// TIA Portal V17 export
// export: Created 2024-08-26T21:10:51.7294849Z, ExportSetting WithDefaults, DisplayName Totally Integrated Automation Portal, DisplayVersion V17 Update 7, DisplayName TIA Portal Openness, DisplayVersion V17 Update 7, DisplayName TIA Portal Version Control Interface, DisplayVersion V17, DisplayName SINAMICS Startdrive Advanced, DisplayVersion V17 SP2, DisplayName SINAMICS Startdrive G110M, G120, G120C, G120D, G120P, G115D, DisplayVersion V17 SP2, DisplayName SINAMICS Startdrive G130, G150, S120, S150, SINAMICS MV, S210, DisplayVersion V17 SP2, DisplayName STEP 7 Professional, DisplayVersion V17 Update 7, DisplayName STEP 7 Safety, DisplayVersion V17 Update 6, DisplayName WinCC Advanced / Unified PC, DisplayVersion V17 Update 7
DATA_BLOCK "DB_MODEL"   // DB5
{ S7_Optimized_Access := 'TRUE' }
VERSION : 0.1
// stored: AutoNumber false, DBAccessibleFromOPCUA true, DBAccessibleFromWebserver true, IsOnlyStoredInLoadMemory false, IsRetainMemResEnabled false, IsWriteProtectedInAS false, MemoryReserve 100
   VAR RETAIN
      "name" : Array[0..32] of String[50];
   END_VAR
   VAR
      day : Int := 6;
      dayText : String := '    11';
      month : Int := 8;
      monthText : String := '     8';
      year : Int := 2012;
      yearReady : String := '2012';
      hour : Int := 17;
      hourText : String := '    17';
      minutes : Int := 30;
      minutesText : String := '    30';
      seconds : Int := 30;
      secondsText : String := '    31';
      active : Array[0..32] of Bool;
   END_VAR
   VAR RETAIN
      datum1 : Array[0..32] of String[50];
      datum2 : Array[0..32] of String[50];
      datum3 : Array[0..32] of String[50];
      datum4 : Array[0..32] of String[50];
      datum5 : Array[0..32] of String[50];
      datum6 : Array[0..32] of String[50];
      datum7 : Array[0..32] of String[50];
   END_VAR
BEGIN
   "name"[0] := 'RH MAN';
   "name"[1] := 'LH MAN';
   "name"[2] := 'RH MAN';
   "name"[3] := '721X';
   "name"[4] := 'STRAP';
   "name"[5] := 'BRACKET';
   "name"[6] := 'FULL FRAME';
   "name"[7..32] := '';
   active[0] := FALSE;
   active[1..6] := TRUE;
   active[7..32] := FALSE;
   datum1[0..2] := 'Z';
   datum1[3] := 'ddd';
   datum1[4..17] := 'Z';
   datum1[18..32] := '';
   datum2[0..17] := '410';
   datum2[18..32] := '';
   datum3[0..17] := '6';
   datum3[18..32] := '';
   datum4[0..2] := 'BACKREST W33A POWER MEMO L6';
   datum4[3] := 'prueba';
   datum4[4] := 'outter trackw33';
   datum4[5..16] := 'BACKREST W33A POWER MEMO L6';
   datum4[17] := 'P42LHNOMEM';
   datum4[18..32] := '';
   datum5[0] := '2389161X-01';
   datum5[1..2] := '2521784';
   datum5[3] := '2389161X-01';
   datum5[4..5] := '2282685X-01';
   datum5[6..16] := '2521784';
   datum5[17] := '2418723X-01';
   datum5[18..32] := '';
   datum6[0..32] := '';
   datum7[0..32] := '';
END_DATA_BLOCK
